// TIA Portal V17 export
// export: Created 2025-06-26T07:49:56.3715127Z, ExportSetting WithDefaults, DisplayName Totally Integrated Automation Portal, DisplayVersion V17 Update 8, DisplayName TIA Portal Openness, DisplayVersion V17 Update 8, DisplayName TIA Portal Version Control Interface, DisplayVersion V17, DisplayName STEP 7 Professional, DisplayVersion V17 Update 8, DisplayName STEP 7 Safety, DisplayVersion V17 Update 6, DisplayName WinCC Advanced, DisplayVersion V17 Update 8
TYPE "stPeriodicRegulator"
// stored: IsFailsafeCompliant false
   STRUCT
      bEnable : Bool;   // 1 = controller enabled, 0 = disabled
      bFault : Bool;   // 1 = controller fault, 0 = ok
      bReset : Bool;   // 1 = reset manual modes, 0 = do nothing
      nMode : USInt;   // 0 = Off, 1 = Auto, 2 = Manual, 3 = Manual Override
      bOutput : Bool;   // 1 = output active
      tOnTime : Time;   // Active time
      tPeriod : Time;   // Repetition time
      tOnTimeElapsed : Time;   // Elapsed time
      tPeriodElapsed : Time;   // Elapsed time
      bManualOverride : Bool;   // 1 = activate override
      bOverrideCmd : Bool;   // 1 = force output on
   END_STRUCT;
END_TYPE
